FUNCTION_BLOCK FifoBuffer
VAR_INPUT
	bOverwrite	: BOOL;
	in 			: IShelfElement;
END_VAR
VAR_OUTPUT
	bOk			: BOOL;
	nCount		: UDINT;
	nLoad		: UDINT;
	out			: IShelfElement;
END_VAR
VAR
	arrBuffer 	: ARRAY[0..MAX_BUFFER_SIZE] OF BYTE; (* Buffer memory used by FB_MemRingBuffer function block *)
	fbBuffer	: FB_MemRingBuffer;
END_VAR
VAR CONSTANT
	MAX_BUFFER_SIZE : UDINT := 1000;
END_VAR

;

ACTION A_Add:
fbBuffer.A_AddTail( pWrite:= ADR( in ),
					cbWrite:= SIZEOF( in ),
					pBuffer:= ADR( arrBuffer ),
					cbBuffer:= SIZEOF( arrBuffer ),
					bOk=> bOk,
					nCount => nCount );


IF NOT bOk THEN (* overflow ? *)
	IF bOverwrite THEN
		fbBuffer.A_RemoveHead(); (* remove one oldest entry *)

		fbBuffer.A_AddTail( bOk => bOk, nCount => nCount );
	END_IF
END_IF



nLoad := (fbBuffer.cbSize * 100) / MAX_BUFFER_SIZE;
END_ACTION

ACTION A_Get:
fbBuffer.A_GetHead( pRead:= ADR( out ),
					cbRead:= SIZEOF( out ),
					pBuffer:= ADR( arrBuffer ),
					cbBuffer:= SIZEOF( arrBuffer ),
					bOk=> bOk,
					nCount => nCount );

nLoad := (fbBuffer.cbSize * 100) / MAX_BUFFER_SIZE;
END_ACTION

ACTION A_Remove:
fbBuffer.A_RemoveHead( 	pRead:= ADR( out ),
						cbRead:= SIZEOF( out ),
						pBuffer:= ADR( arrBuffer ),
						cbBuffer:= SIZEOF( arrBuffer ),
						bOk=> bOk,
						nCount => nCount );

nLoad := (fbBuffer.cbSize * 100) / MAX_BUFFER_SIZE;
END_ACTION

ACTION A_Reset:
MEMSET( ADR( arrBuffer ), 0, SIZEOF( arrBuffer ) ); (* reset (optional) internal buffer *)

fbBuffer.A_Reset( 	bOk=> bOk,
					nCount => nCount );

nLoad := (fbBuffer.cbSize * 100) / MAX_BUFFER_SIZE;
END_ACTION

END_FUNCTION_BLOCK

(* stored: Version 1.1.0.1
   POU FifoBuffer: Id {68aab722-1c15-4a1c-8558-70d8155fb516}, SpecialFunc None
   Action A_Add: Id {a7dab110-6508-416f-acc6-ce74c3eacfc5}
   Action A_Get: Id {6033ce75-8df1-402c-b27d-509c03464659}
   Action A_Remove: Id {53dc8178-a4b4-4f80-9c5f-a4c816f0e571}
   Action A_Reset: Id {13e425e4-714d-4cfe-9858-15b661921577} *)
